TEXTLIST TextList_Type_Etape
  0 = 'Aucun' | FR: 'Aucun' | EN: 'None'
  1 = '' | FR: 'Pompage chambre' | EN: 'Chamber pumping'
  2 = '' | FR: 'Isolement chambre' | EN: 'Chamber standby'
  3 = '' | FR: 'Marche pompes chambre' | EN: 'Chamber pumps start'
  4 = '' | FR: 'Arrêt pompes chambre' | EN: 'Chamber pumps stop'
  5 = '' | FR: 'Régénération pompe cryogénique' | EN: 'Cryo Pump regeneration'
  6 = '' | FR: 'Ventilation chambre' | EN: 'Chamber venting'
  7 = '' | FR: "Point d'arrêt" | EN: 'Break point'
  8 = '' | FR: 'Evaporation' | EN: 'Evaporation'
  9 = '' | FR: 'Synchronisation horaire' | EN: 'Time synchronization'
  10 = '' | FR: 'Temporisation' | EN: 'Timer'
  11 = '' | FR: 'Rotation PS' | EN: 'SH Rotation'
  12 = '' | FR: 'Arrêt rotation PS' | EN: 'SH Stop Rotation'
  13 = '' | FR: 'Effluvage' | EN: 'Glow discharge'
  14 = '' | FR: 'Test de remontée de pression' | EN: 'Pressure rise test'
  15 = '' | FR: 'Arrêt procédé' | EN: 'Stopping process'
  16 = '' | FR: 'Boucle/Saut' | EN: 'Loop/Skip'
  17 = '' | FR: 'Lancement Eco-veille' | EN: 'Start Eco-sleep'
  18 = '' | FR: 'Arrêt Eco-veille' | EN: 'Stop Eco-sleep'
  19 = '' | FR: 'Régénération partielle cryo' | EN: 'Cryo pump partial regeneration'
   = ''
END_TEXTLIST

(* stored: Version 1.1.0.1, ProductVersion 3.1.4024.10
   TextList TextList_Type_Etape: Id {d19fa78e-07bb-4c51-a5d8-3293143f07ca} *)
